FUNCTION_BLOCK PrevCurrState (* Basic Function Block Type *)
  (* Standard: 61499-2 *)
  (* Version 0.0, 6/11/2026, Schneider Electric, Template *)
  PACKAGE SE.Nereda;
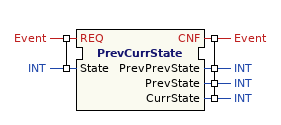
  EVENT_INPUT
    REQ WITH State; (* Normal Execution Request *)
  END_EVENT
  EVENT_OUTPUT
    CNF WITH PrevPrevState, PrevState, CurrState; (* Execution Confirmation *)
  END_EVENT
  VAR_INPUT
    State : INT;
  END_VAR
  VAR_OUTPUT
    PrevPrevState : INT;
    PrevState : INT;
    CurrState : INT;
  END_VAR
  VAR
    InTable : ARRAY [0..2] OF INT;
  END_VAR
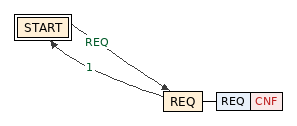
  EC_STATES
    START; (* Initial State *)
    REQ : REQ -> CNF; (* Normal execution *)
  END_STATES
  EC_TRANSITIONS
    START TO REQ := REQ;
    REQ TO START := 1;
  END_TRANSITIONS
  ALGORITHM REQ IN ST: (* Normally executed algorithm *)
;

IF CurrState <> State THEN
	InTable[2] := InTable[1];
	InTable[1] := InTable[0];
	InTable[0] := State;
END_IF;

PrevPrevState := InTable[2];
PrevState := InTable[1];
CurrState := InTable[0];
  END_ALGORITHM
END_FUNCTION_BLOCK
